{attribute 'GeneratedUsingTerminal: EL6001-0000-0020'}
{attribute addProperty BoxType "EL6001-0000-0020"}
{attribute addProperty Id "COM_ext_inputsAT %I*COM_ext_inputs_1F197B20108COM_ext_outputsAT %Q*COM_ext_outputs_54D54ACC105WcStateAT %I*WcState_9091E0EB2InfoDataAT %I*InfoData_94A18F5E2"}
{attribute addProperty CRC "3558919390"}
{attribute addProperty Size "217"}
TYPE EL6001_D420CCDE EXTENDS EtcSlaveTerminalBase_947E5A46 :
STRUCT
	{attribute addProperty Name "COM_ext_inputs"}
	COM_ext_inputs : COM_ext_inputs_1F197B20;
	{attribute addProperty Name "COM_ext_outputs"}
	COM_ext_outputs : COM_ext_outputs_54D54ACC;
	{attribute addProperty Name "WcState"}
	WcState : WcState_9091E0EB;
	{attribute addProperty Name "InfoData"}
	InfoData : InfoData_94A18F5E;
END_STRUCT
END_TYPE

(* stored: Version 1.2.0.0, ProductVersion 3.1.4024.9
   DUT EL6001_D420CCDE: Id {c1700b35-ea40-4e35-9496-585b730e3571} *)
